Xinje XCPPro project, PLC1: XC5-32-4PLS (software 3.3q 2017-01-03)

PROGRAM Ladder

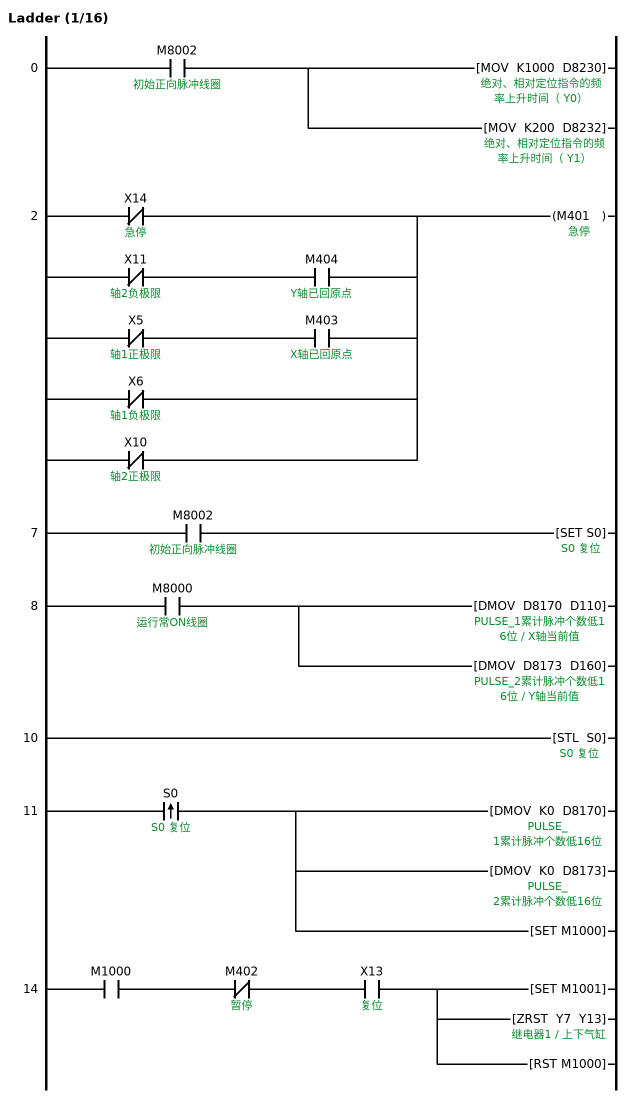
LD     M8002	; 初始正向脉冲线圈
MOV    K1000 D8230	; 绝对、相对定位指令的频率上升时间（ Y0）
MOV    K200 D8232	; 绝对、相对定位指令的频率上升时间（ Y1）
LDI    X14	; 急停
LDI    X11	; 轴2负极限
AND    M404	; Y轴已回原点
ORB
LDI    X5	; 轴1正极限
AND    M403	; X轴已回原点
ORB
ORI    X6	; 轴1负极限
ORI    X10	; 轴2正极限
OUT    M401	; 急停
LD     M8002	; 初始正向脉冲线圈
SET    S0	; S0 复位
LD     M8000	; 运行常ON线圈
DMOV   D8170 D110	; PULSE_1累计脉冲个数低16位 / X轴当前值
DMOV   D8173 D160	; PULSE_2累计脉冲个数低16位 / Y轴当前值
STL    S0	; S0 复位
LDP    S0	; S0 复位
DMOV   K0 D8170	; PULSE_1累计脉冲个数低16位
DMOV   K0 D8173	; PULSE_2累计脉冲个数低16位
SET    M1000
LD     M1000
ANI    M402	; 暂停
AND    X13	; 复位
SET    M1001
ZRST   Y7 Y13	; 继电器1 / 上下气缸
RST    M1000

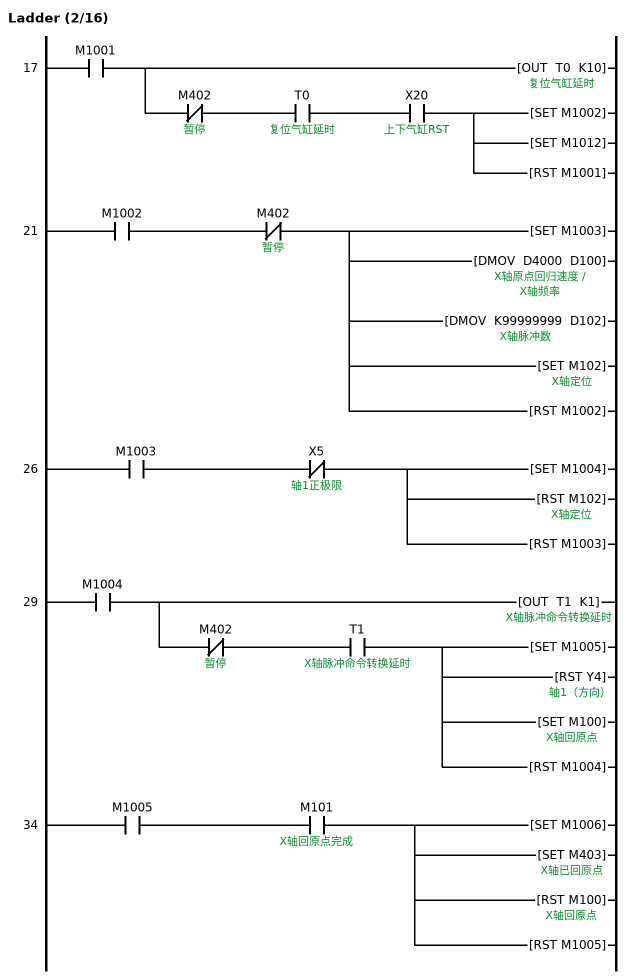
LD     M1001
OUT    T0 K10	; 复位气缸延时
ANI    M402	; 暂停
AND    T0	; 复位气缸延时
AND    X20	; 上下气缸RST
SET    M1002
SET    M1012
RST    M1001
LD     M1002
ANI    M402	; 暂停
SET    M1003
DMOV   D4000 D100	; X轴原点回归速度 / X轴频率
DMOV   K99999999 D102	; X轴脉冲数
SET    M102	; X轴定位
RST    M1002
LD     M1003
ANI    X5	; 轴1正极限
SET    M1004
RST    M102	; X轴定位
RST    M1003
LD     M1004
OUT    T1 K1	; X轴脉冲命令转换延时
ANI    M402	; 暂停
AND    T1	; X轴脉冲命令转换延时
SET    M1005
RST    Y4	; 轴1（方向）
SET    M100	; X轴回原点
RST    M1004
LD     M1005
AND    M101	; X轴回原点完成
SET    M1006
SET    M403	; X轴已回原点
RST    M100	; X轴回原点
RST    M1005

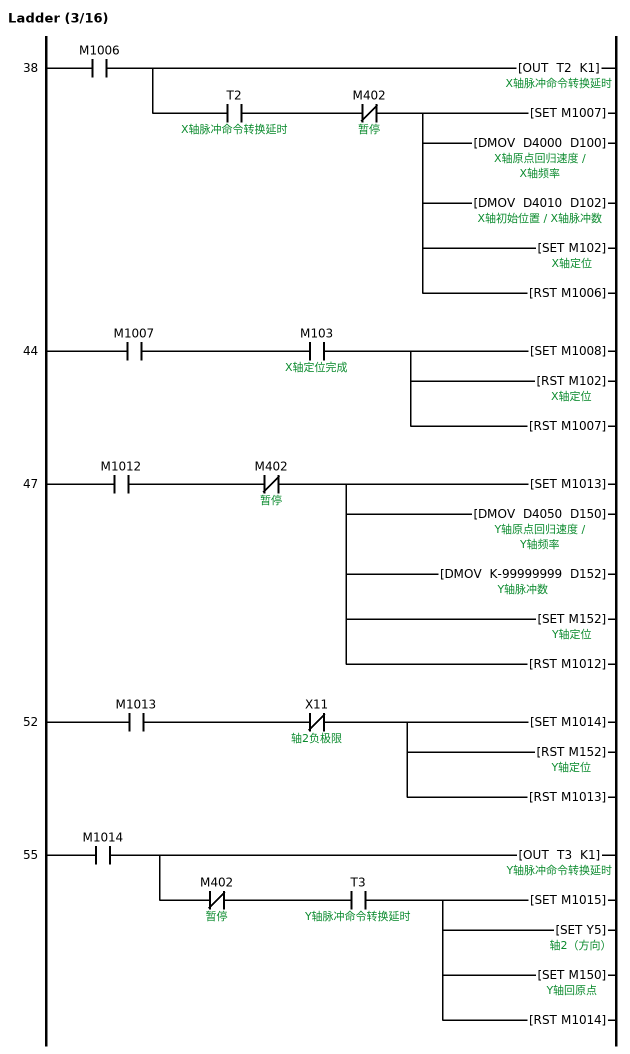
LD     M1006
OUT    T2 K1	; X轴脉冲命令转换延时
AND    T2	; X轴脉冲命令转换延时
ANI    M402	; 暂停
SET    M1007
DMOV   D4000 D100	; X轴原点回归速度 / X轴频率
DMOV   D4010 D102	; X轴初始位置 / X轴脉冲数
SET    M102	; X轴定位
RST    M1006
LD     M1007
AND    M103	; X轴定位完成
SET    M1008
RST    M102	; X轴定位
RST    M1007
LD     M1012
ANI    M402	; 暂停
SET    M1013
DMOV   D4050 D150	; Y轴原点回归速度 / Y轴频率
DMOV   K-99999999 D152	; Y轴脉冲数
SET    M152	; Y轴定位
RST    M1012
LD     M1013
ANI    X11	; 轴2负极限
SET    M1014
RST    M152	; Y轴定位
RST    M1013
LD     M1014
OUT    T3 K1	; Y轴脉冲命令转换延时
ANI    M402	; 暂停
AND    T3	; Y轴脉冲命令转换延时
SET    M1015
SET    Y5	; 轴2（方向）
SET    M150	; Y轴回原点
RST    M1014

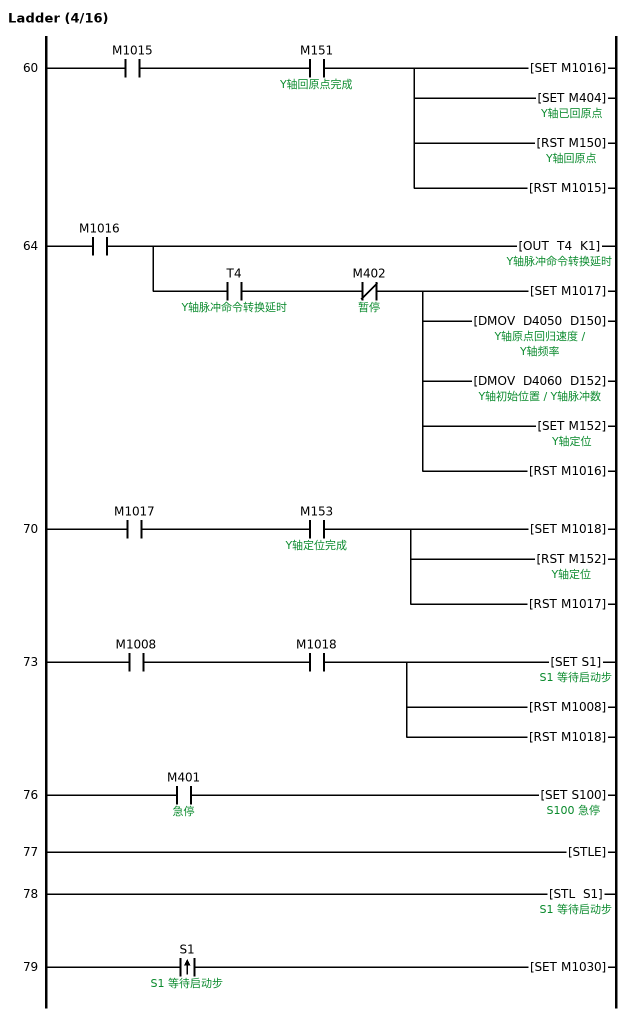
LD     M1015
AND    M151	; Y轴回原点完成
SET    M1016
SET    M404	; Y轴已回原点
RST    M150	; Y轴回原点
RST    M1015
LD     M1016
OUT    T4 K1	; Y轴脉冲命令转换延时
AND    T4	; Y轴脉冲命令转换延时
ANI    M402	; 暂停
SET    M1017
DMOV   D4050 D150	; Y轴原点回归速度 / Y轴频率
DMOV   D4060 D152	; Y轴初始位置 / Y轴脉冲数
SET    M152	; Y轴定位
RST    M1016
LD     M1017
AND    M153	; Y轴定位完成
SET    M1018
RST    M152	; Y轴定位
RST    M1017
LD     M1008
AND    M1018
SET    S1	; S1 等待启动步
RST    M1008
RST    M1018
LD     M401	; 急停
SET    S100	; S100 急停
STLE
STL    S1	; S1 等待启动步
LDP    S1	; S1 等待启动步
SET    M1030

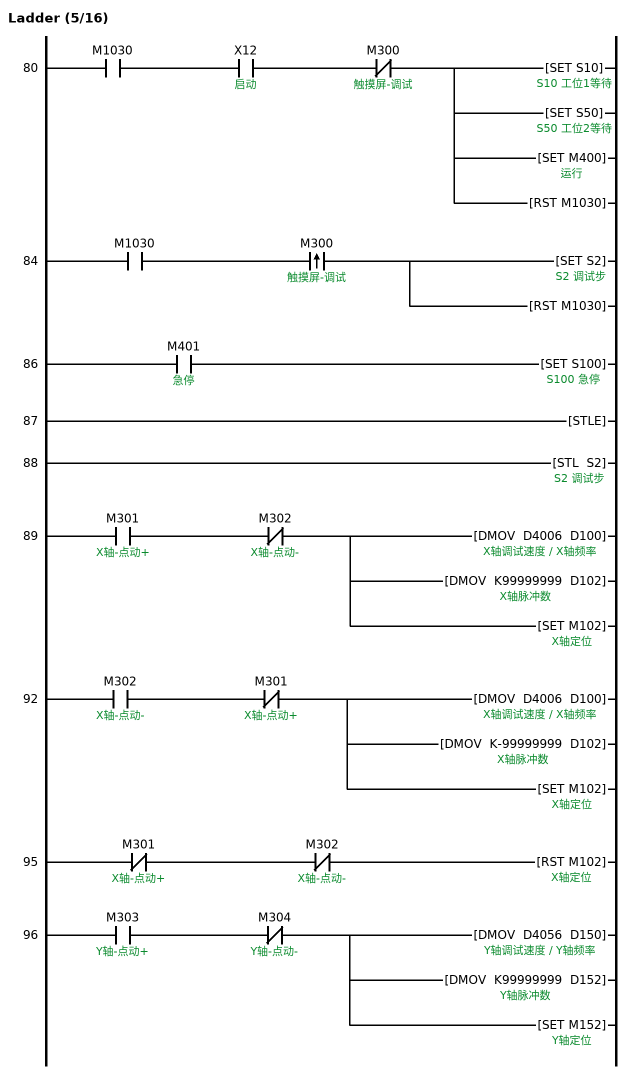
LD     M1030
AND    X12	; 启动
ANI    M300	; 触摸屏-调试
SET    S10	; S10 工位1等待
SET    S50	; S50 工位2等待
SET    M400	; 运行
RST    M1030
LD     M1030
ANDP   M300	; 触摸屏-调试
SET    S2	; S2 调试步
RST    M1030
LD     M401	; 急停
SET    S100	; S100 急停
STLE
STL    S2	; S2 调试步
LD     M301	; X轴-点动+
ANI    M302	; X轴-点动-
DMOV   D4006 D100	; X轴调试速度 / X轴频率
DMOV   K99999999 D102	; X轴脉冲数
SET    M102	; X轴定位
LD     M302	; X轴-点动-
ANI    M301	; X轴-点动+
DMOV   D4006 D100	; X轴调试速度 / X轴频率
DMOV   K-99999999 D102	; X轴脉冲数
SET    M102	; X轴定位
LDI    M301	; X轴-点动+
ANI    M302	; X轴-点动-
RST    M102	; X轴定位
LD     M303	; Y轴-点动+
ANI    M304	; Y轴-点动-
DMOV   D4056 D150	; Y轴调试速度 / Y轴频率
DMOV   K99999999 D152	; Y轴脉冲数
SET    M152	; Y轴定位

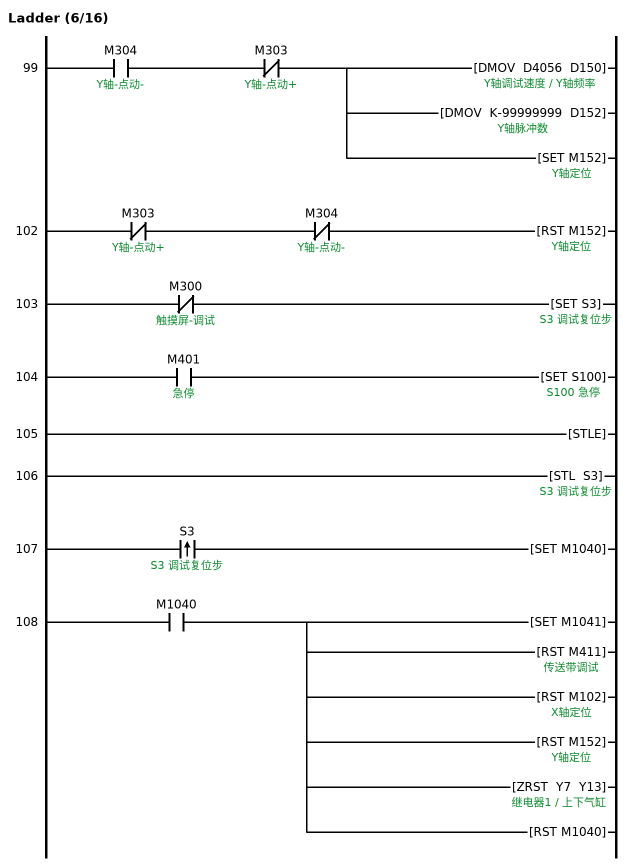
LD     M304	; Y轴-点动-
ANI    M303	; Y轴-点动+
DMOV   D4056 D150	; Y轴调试速度 / Y轴频率
DMOV   K-99999999 D152	; Y轴脉冲数
SET    M152	; Y轴定位
LDI    M303	; Y轴-点动+
ANI    M304	; Y轴-点动-
RST    M152	; Y轴定位
LDI    M300	; 触摸屏-调试
SET    S3	; S3 调试复位步
LD     M401	; 急停
SET    S100	; S100 急停
STLE
STL    S3	; S3 调试复位步
LDP    S3	; S3 调试复位步
SET    M1040
LD     M1040
SET    M1041
RST    M411	; 传送带调试
RST    M102	; X轴定位
RST    M152	; Y轴定位
ZRST   Y7 Y13	; 继电器1 / 上下气缸
RST    M1040

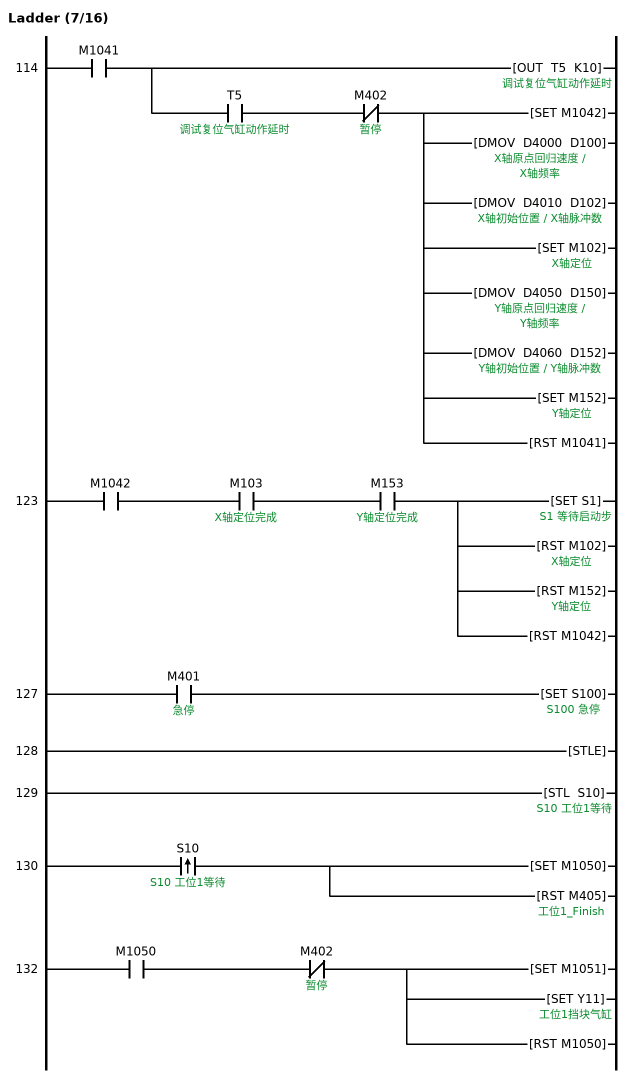
LD     M1041
OUT    T5 K10	; 调试复位气缸动作延时
AND    T5	; 调试复位气缸动作延时
ANI    M402	; 暂停
SET    M1042
DMOV   D4000 D100	; X轴原点回归速度 / X轴频率
DMOV   D4010 D102	; X轴初始位置 / X轴脉冲数
SET    M102	; X轴定位
DMOV   D4050 D150	; Y轴原点回归速度 / Y轴频率
DMOV   D4060 D152	; Y轴初始位置 / Y轴脉冲数
SET    M152	; Y轴定位
RST    M1041
LD     M1042
AND    M103	; X轴定位完成
AND    M153	; Y轴定位完成
SET    S1	; S1 等待启动步
RST    M102	; X轴定位
RST    M152	; Y轴定位
RST    M1042
LD     M401	; 急停
SET    S100	; S100 急停
STLE
STL    S10	; S10 工位1等待
LDP    S10	; S10 工位1等待
SET    M1050
RST    M405	; 工位1_Finish
LD     M1050
ANI    M402	; 暂停
SET    M1051
SET    Y11	; 工位1挡块气缸
RST    M1050

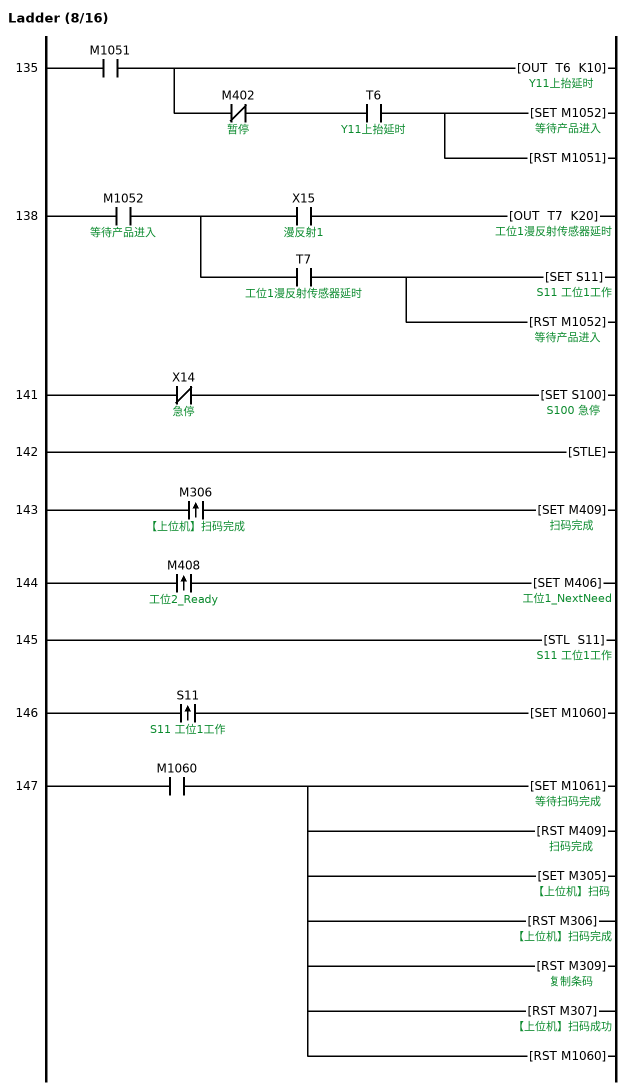
LD     M1051
OUT    T6 K10	; Y11上抬延时
ANI    M402	; 暂停
AND    T6	; Y11上抬延时
SET    M1052	; 等待产品进入
RST    M1051
LD     M1052	; 等待产品进入
MPS
AND    X15	; 漫反射1
OUT    T7 K20	; 工位1漫反射传感器延时
MPP
AND    T7	; 工位1漫反射传感器延时
SET    S11	; S11 工位1工作
RST    M1052	; 等待产品进入
LDI    X14	; 急停
SET    S100	; S100 急停
STLE
LDP    M306	; 【上位机】扫码完成
SET    M409	; 扫码完成
LDP    M408	; 工位2_Ready
SET    M406	; 工位1_NextNeed
STL    S11	; S11 工位1工作
LDP    S11	; S11 工位1工作
SET    M1060
LD     M1060
SET    M1061	; 等待扫码完成
RST    M409	; 扫码完成
SET    M305	; 【上位机】扫码
RST    M306	; 【上位机】扫码完成
RST    M309	; 复制条码
RST    M307	; 【上位机】扫码成功
RST    M1060

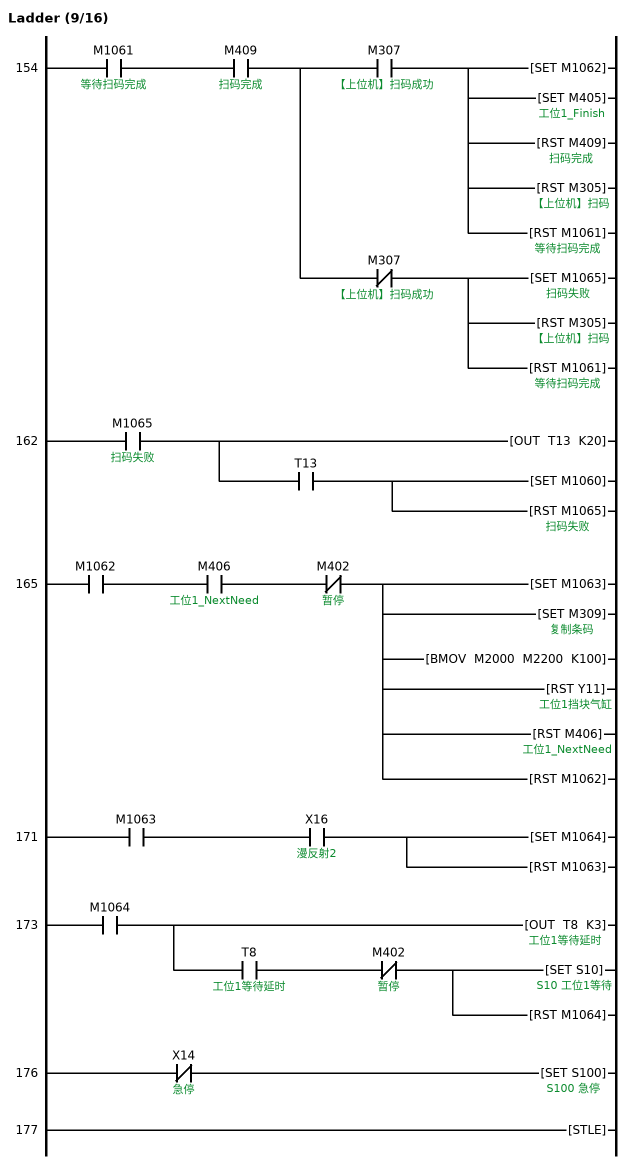
LD     M1061	; 等待扫码完成
AND    M409	; 扫码完成
MPS
AND    M307	; 【上位机】扫码成功
SET    M1062
SET    M405	; 工位1_Finish
RST    M409	; 扫码完成
RST    M305	; 【上位机】扫码
RST    M1061	; 等待扫码完成
MPP
ANI    M307	; 【上位机】扫码成功
SET    M1065	; 扫码失败
RST    M305	; 【上位机】扫码
RST    M1061	; 等待扫码完成
LD     M1065	; 扫码失败
OUT    T13 K20
AND    T13
SET    M1060
RST    M1065	; 扫码失败
LD     M1062
AND    M406	; 工位1_NextNeed
ANI    M402	; 暂停
SET    M1063
SET    M309	; 复制条码
BMOV   M2000 M2200 K100
RST    Y11	; 工位1挡块气缸
RST    M406	; 工位1_NextNeed
RST    M1062
LD     M1063
AND    X16	; 漫反射2
SET    M1064
RST    M1063
LD     M1064
OUT    T8 K3	; 工位1等待延时
AND    T8	; 工位1等待延时
ANI    M402	; 暂停
SET    S10	; S10 工位1等待
RST    M1064
LDI    X14	; 急停
SET    S100	; S100 急停
STLE

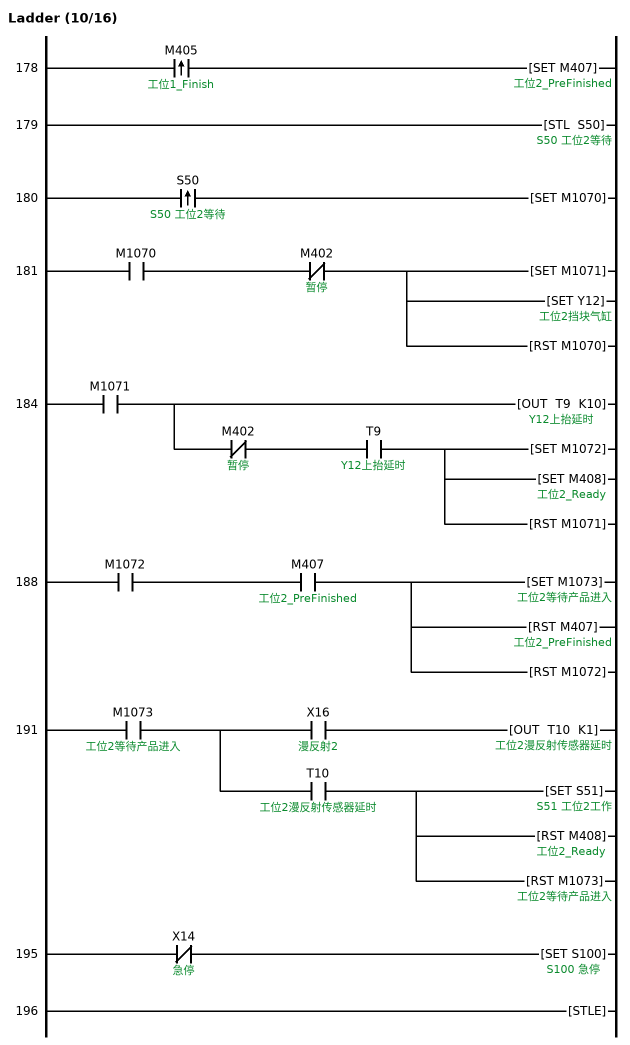
LDP    M405	; 工位1_Finish
SET    M407	; 工位2_PreFinished
STL    S50	; S50 工位2等待
LDP    S50	; S50 工位2等待
SET    M1070
LD     M1070
ANI    M402	; 暂停
SET    M1071
SET    Y12	; 工位2挡块气缸
RST    M1070
LD     M1071
OUT    T9 K10	; Y12上抬延时
ANI    M402	; 暂停
AND    T9	; Y12上抬延时
SET    M1072
SET    M408	; 工位2_Ready
RST    M1071
LD     M1072
AND    M407	; 工位2_PreFinished
SET    M1073	; 工位2等待产品进入
RST    M407	; 工位2_PreFinished
RST    M1072
LD     M1073	; 工位2等待产品进入
MPS
AND    X16	; 漫反射2
OUT    T10 K1	; 工位2漫反射传感器延时
MPP
AND    T10	; 工位2漫反射传感器延时
SET    S51	; S51 工位2工作
RST    M408	; 工位2_Ready
RST    M1073	; 工位2等待产品进入
LDI    X14	; 急停
SET    S100	; S100 急停
STLE

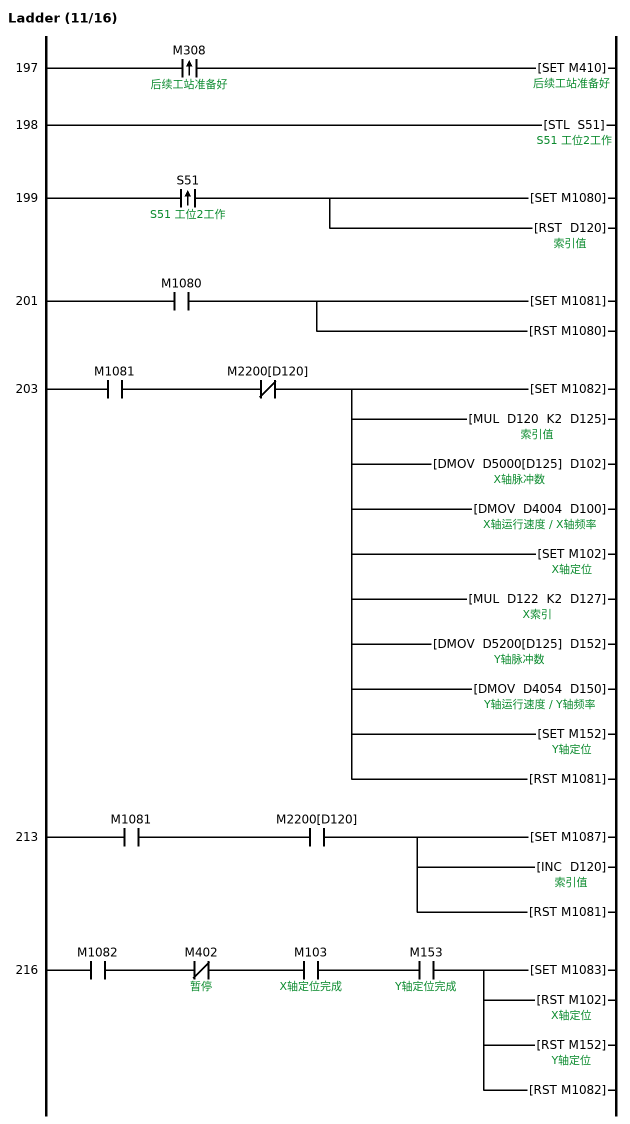
LDP    M308	; 后续工站准备好
SET    M410	; 后续工站准备好
STL    S51	; S51 工位2工作
LDP    S51	; S51 工位2工作
SET    M1080
RST    D120	; 索引值
LD     M1080
SET    M1081
RST    M1080
LD     M1081
ANI    M2200[D120]
SET    M1082
MUL    D120 K2 D125	; 索引值
DMOV   D5000[D125] D102	; X轴脉冲数
DMOV   D4004 D100	; X轴运行速度 / X轴频率
SET    M102	; X轴定位
MUL    D122 K2 D127	; X索引
DMOV   D5200[D125] D152	; Y轴脉冲数
DMOV   D4054 D150	; Y轴运行速度 / Y轴频率
SET    M152	; Y轴定位
RST    M1081
LD     M1081
AND    M2200[D120]
SET    M1087
INC    D120	; 索引值
RST    M1081
LD     M1082
ANI    M402	; 暂停
AND    M103	; X轴定位完成
AND    M153	; Y轴定位完成
SET    M1083
RST    M102	; X轴定位
RST    M152	; Y轴定位
RST    M1082

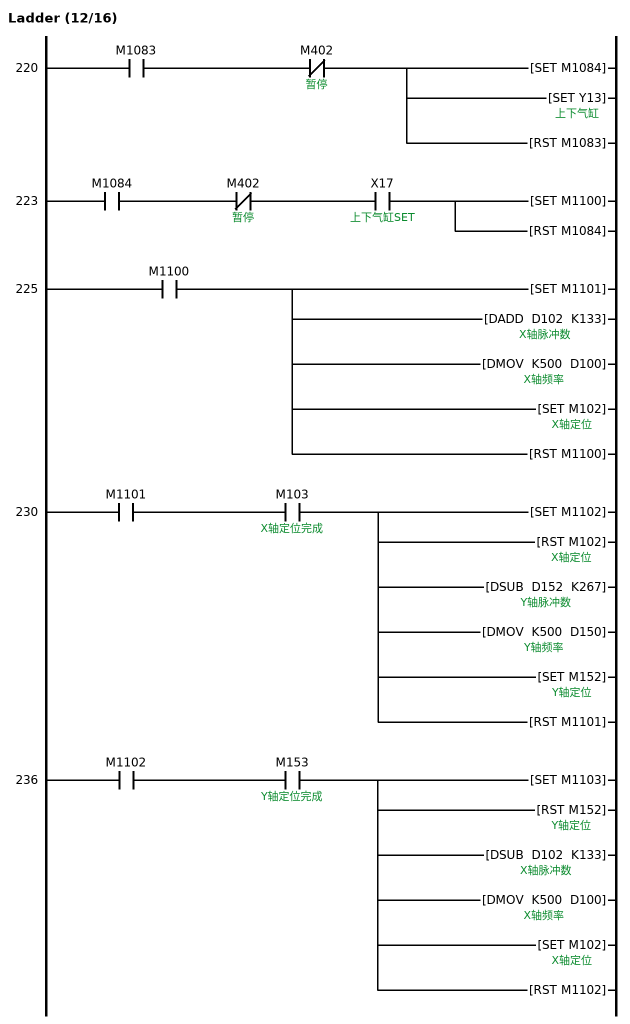
LD     M1083
ANI    M402	; 暂停
SET    M1084
SET    Y13	; 上下气缸
RST    M1083
LD     M1084
ANI    M402	; 暂停
AND    X17	; 上下气缸SET
SET    M1100
RST    M1084
LD     M1100
SET    M1101
DADD   D102 K133	; X轴脉冲数
DMOV   K500 D100	; X轴频率
SET    M102	; X轴定位
RST    M1100
LD     M1101
AND    M103	; X轴定位完成
SET    M1102
RST    M102	; X轴定位
DSUB   D152 K267	; Y轴脉冲数
DMOV   K500 D150	; Y轴频率
SET    M152	; Y轴定位
RST    M1101
LD     M1102
AND    M153	; Y轴定位完成
SET    M1103
RST    M152	; Y轴定位
DSUB   D102 K133	; X轴脉冲数
DMOV   K500 D100	; X轴频率
SET    M102	; X轴定位
RST    M1102

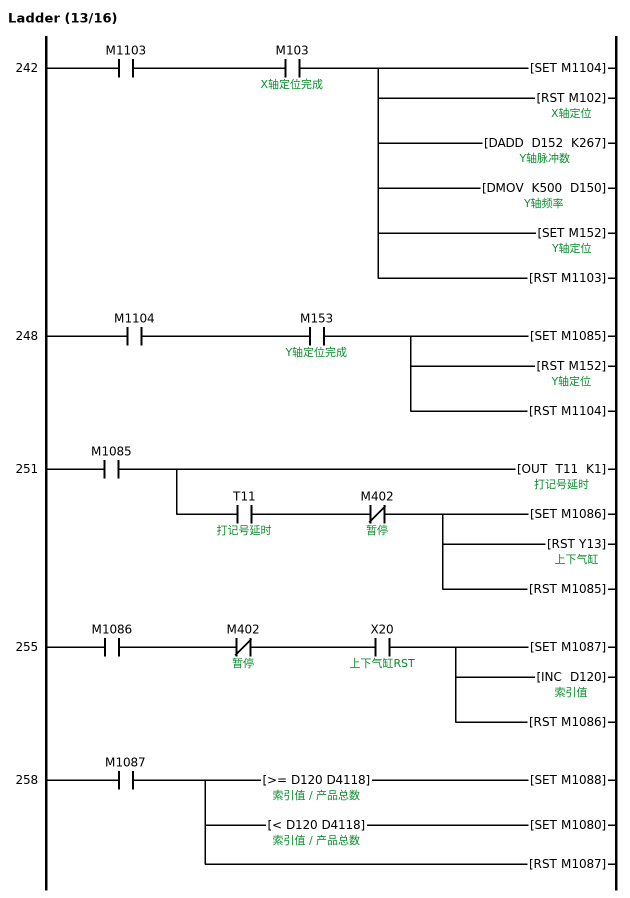
LD     M1103
AND    M103	; X轴定位完成
SET    M1104
RST    M102	; X轴定位
DADD   D152 K267	; Y轴脉冲数
DMOV   K500 D150	; Y轴频率
SET    M152	; Y轴定位
RST    M1103
LD     M1104
AND    M153	; Y轴定位完成
SET    M1085
RST    M152	; Y轴定位
RST    M1104
LD     M1085
OUT    T11 K1	; 打记号延时
AND    T11	; 打记号延时
ANI    M402	; 暂停
SET    M1086
RST    Y13	; 上下气缸
RST    M1085
LD     M1086
ANI    M402	; 暂停
AND    X20	; 上下气缸RST
SET    M1087
INC    D120	; 索引值
RST    M1086
LD     M1087
MPS
AND>=  D120 D4118	; 索引值 / 产品总数
SET    M1088
MRD
AND<   D120 D4118	; 索引值 / 产品总数
SET    M1080
MPP
RST    M1087

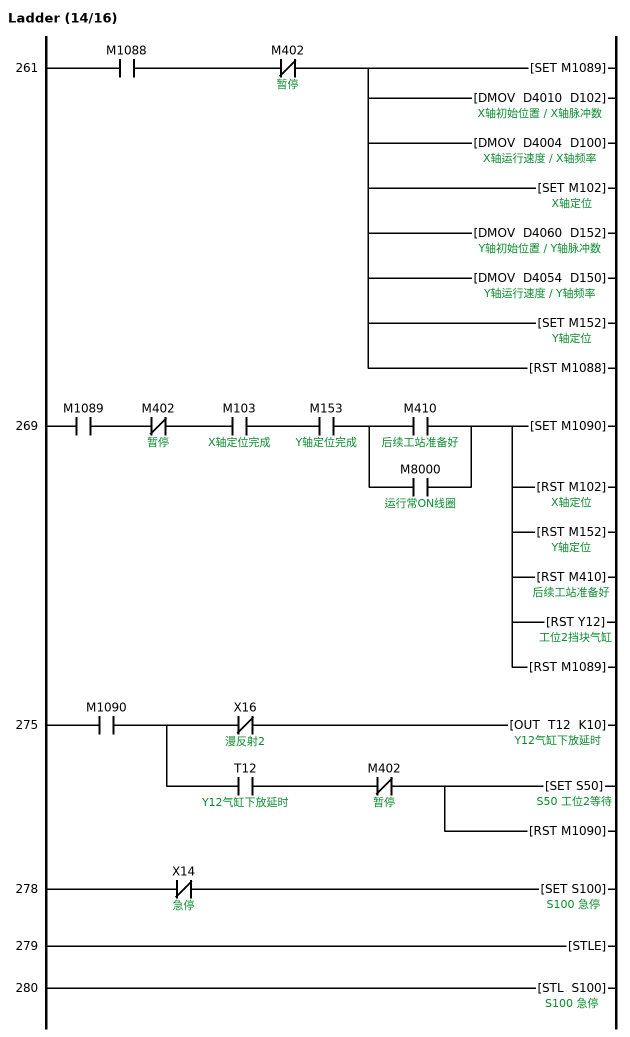
LD     M1088
ANI    M402	; 暂停
SET    M1089
DMOV   D4010 D102	; X轴初始位置 / X轴脉冲数
DMOV   D4004 D100	; X轴运行速度 / X轴频率
SET    M102	; X轴定位
DMOV   D4060 D152	; Y轴初始位置 / Y轴脉冲数
DMOV   D4054 D150	; Y轴运行速度 / Y轴频率
SET    M152	; Y轴定位
RST    M1088
LD     M1089
ANI    M402	; 暂停
AND    M103	; X轴定位完成
AND    M153	; Y轴定位完成
LD     M410	; 后续工站准备好
OR     M8000	; 运行常ON线圈
ANB
SET    M1090
RST    M102	; X轴定位
RST    M152	; Y轴定位
RST    M410	; 后续工站准备好
RST    Y12	; 工位2挡块气缸
RST    M1089
LD     M1090
MPS
ANI    X16	; 漫反射2
OUT    T12 K10	; Y12气缸下放延时
MPP
AND    T12	; Y12气缸下放延时
ANI    M402	; 暂停
SET    S50	; S50 工位2等待
RST    M1090
LDI    X14	; 急停
SET    S100	; S100 急停
STLE
STL    S100	; S100 急停

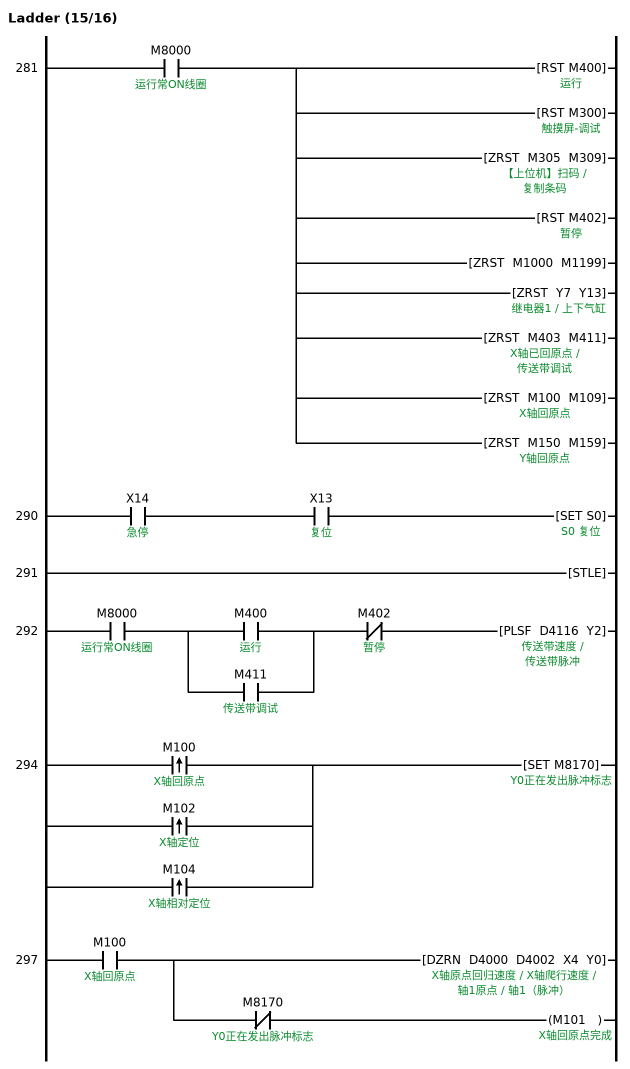
LD     M8000	; 运行常ON线圈
RST    M400	; 运行
RST    M300	; 触摸屏-调试
ZRST   M305 M309	; 【上位机】扫码 / 复制条码
RST    M402	; 暂停
ZRST   M1000 M1199
ZRST   Y7 Y13	; 继电器1 / 上下气缸
ZRST   M403 M411	; X轴已回原点 / 传送带调试
ZRST   M100 M109	; X轴回原点
ZRST   M150 M159	; Y轴回原点
LD     X14	; 急停
AND    X13	; 复位
SET    S0	; S0 复位
STLE
LD     M8000	; 运行常ON线圈
LD     M400	; 运行
OR     M411	; 传送带调试
ANB
ANI    M402	; 暂停
PLSF   D4116 Y2	; 传送带速度 / 传送带脉冲
LDP    M100	; X轴回原点
ORP    M102	; X轴定位
ORP    M104	; X轴相对定位
SET    M8170	; Y0正在发出脉冲标志
LD     M100	; X轴回原点
DZRN   D4000 D4002 X4 Y0	; X轴原点回归速度 / X轴爬行速度 / 轴1原点 / 轴1（脉冲）
ANI    M8170	; Y0正在发出脉冲标志
OUT    M101	; X轴回原点完成

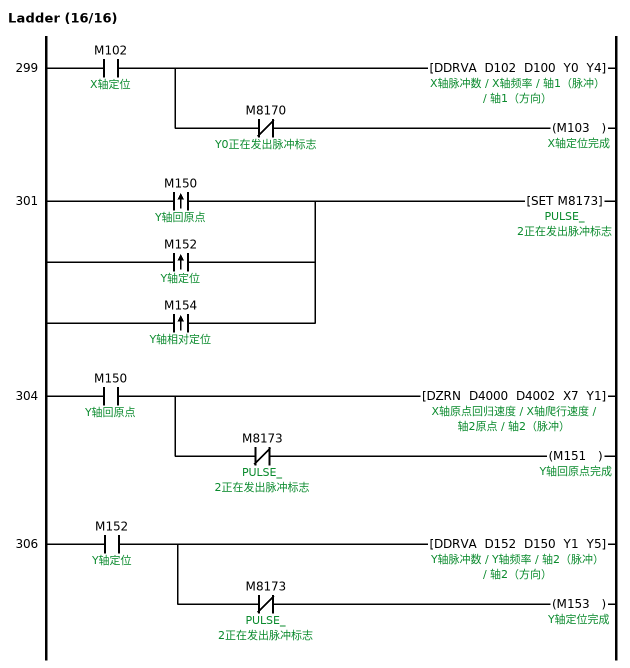
LD     M102	; X轴定位
DDRVA  D102 D100 Y0 Y4	; X轴脉冲数 / X轴频率 / 轴1（脉冲） / 轴1（方向）
ANI    M8170	; Y0正在发出脉冲标志
OUT    M103	; X轴定位完成
LDP    M150	; Y轴回原点
ORP    M152	; Y轴定位
ORP    M154	; Y轴相对定位
SET    M8173	; PULSE_2正在发出脉冲标志
LD     M150	; Y轴回原点
DZRN   D4000 D4002 X7 Y1	; X轴原点回归速度 / X轴爬行速度 / 轴2原点 / 轴2（脉冲）
ANI    M8173	; PULSE_2正在发出脉冲标志
OUT    M151	; Y轴回原点完成
LD     M152	; Y轴定位
DDRVA  D152 D150 Y1 Y5	; Y轴脉冲数 / Y轴频率 / 轴2（脉冲） / 轴2（方向）
ANI    M8173	; PULSE_2正在发出脉冲标志
OUT    M153	; Y轴定位完成

COMMENTS (devices not used above)
Y10	继电器2
M105	X轴相对定位完成
M155	Y轴相对定位完成
D104	X轴频率1
D106	X轴脉冲数1
D154	Y轴频率1
D156	Y轴脉冲数1
D4052	Y轴爬行速度
D4100	X1
D4102	Y1
D4104	X2
D4106	Y2
D4108	X3
D4110	Y3
D4112	X数
D4114	Y数
D5000	X轴点阵1
D5002	X轴点阵2
D5004	X轴点阵3
D5006	X轴点阵4
D5008	X轴点阵5
D5010	X轴点阵6
D5012	X轴点阵7
D5014	X轴点阵8
D5016	X轴点阵9
D5018	X轴点阵10
D5020	X轴点阵11
D5022	X轴点阵12
D5024	X轴点阵13
D5026	X轴点阵14
D5028	X轴点阵15
D5030	X轴点阵16
D5032	X轴点阵17
D5034	X轴点阵18
D5036	X轴点阵19
D5038	X轴点阵20
D5040	X轴点阵21
D5042	X轴点阵22
D5044	X轴点阵23
D5046	X轴点阵24
D5048	X轴点阵25
D5050	X轴点阵26
D5052	X轴点阵27
D5054	X轴点阵28
D5056	X轴点阵29
D5058	X轴点阵30
D5060	X轴点阵31
D5062	X轴点阵32
D5064	X轴点阵33
D5066	X轴点阵34
D5068	X轴点阵35
D5070	X轴点阵36
D5072	X轴点阵37
D5074	X轴点阵38
D5076	X轴点阵39
D5078	X轴点阵40
D5080	X轴点阵41
D5082	X轴点阵42
D5084	X轴点阵43
D5086	X轴点阵44
D5088	X轴点阵45
D5090	X轴点阵46
D5092	X轴点阵47
D5094	X轴点阵48
D5096	X轴点阵49
D5098	X轴点阵50
D5100	X轴点阵51
D5102	X轴点阵52
D5104	X轴点阵53
D5106	X轴点阵54
D5108	X轴点阵55
D5110	X轴点阵56
D5112	X轴点阵57
D5114	X轴点阵58
D5116	X轴点阵59
D5118	X轴点阵60
D5200	Y轴点阵1
D5202	Y轴点阵2
D5204	Y轴点阵3
D5206	Y轴点阵4
D5208	Y轴点阵5
D5210	Y轴点阵6
D5212	Y轴点阵7
D5214	Y轴点阵8
D5216	Y轴点阵9
D5218	Y轴点阵10
D5220	Y轴点阵11
D5222	Y轴点阵12
D5224	Y轴点阵13
D5226	Y轴点阵14
D5228	Y轴点阵15
D5230	Y轴点阵16
D5232	Y轴点阵17
D5234	Y轴点阵18
D5236	Y轴点阵19
D5238	Y轴点阵20
D5240	Y轴点阵21
D5242	Y轴点阵22
D5244	Y轴点阵23
D5246	Y轴点阵24
D5248	Y轴点阵25
D5250	Y轴点阵26
D5252	Y轴点阵27
D5254	Y轴点阵28
D5256	Y轴点阵29
D5258	Y轴点阵30
D5260	Y轴点阵31
D5262	Y轴点阵32
D5264	Y轴点阵33
D5266	Y轴点阵34
D5268	Y轴点阵35
D5270	Y轴点阵36
D5272	Y轴点阵37
D5274	Y轴点阵38
D5276	Y轴点阵39
D5278	Y轴点阵40
D5280	Y轴点阵41
D5282	Y轴点阵42
D5284	Y轴点阵43
D5286	Y轴点阵44
D5288	Y轴点阵45
D5290	Y轴点阵46
D5292	Y轴点阵47
D5294	Y轴点阵48
D5296	Y轴点阵49
D5298	Y轴点阵50
D5300	Y轴点阵51
D5302	Y轴点阵52
D5304	Y轴点阵53
D5306	Y轴点阵54
D5308	Y轴点阵55
D5310	Y轴点阵56
D5312	Y轴点阵57
D5314	Y轴点阵58
D5316	Y轴点阵59
D5318	Y轴点阵60